// TIA Portal V15.1 export
// export: Created 2024-06-21T08:41:23.1994164Z, ExportSetting WithDefaults, DisplayName Totally Integrated Automation Portal, DisplayVersion V15.1 Update 5, DisplayName TIA Portal Openness, DisplayVersion V15.1 Update 5, DisplayName SINAMICS Startdrive Advanced, DisplayVersion V15.1, DisplayName G130, G150, S120, S150, SINAMICS MV, S210, DisplayVersion V15.1, DisplayName G110M, G120, G120C, G120D, G120P, DisplayVersion V15.1, DisplayName STEP 7 Professional, DisplayVersion V15.1 Update 5, DisplayName STEP 7 Safety, DisplayVersion V15.1, DisplayName WinCC Professional, DisplayVersion V15.1 Update 5, DisplayName SIMATIC Visualization Architect, DisplayVersion V15.1
FUNCTION "209210ZS01" : Void   // FC320, FBD
TITLE = 209210ZS01 Safety zone
{ S7_Optimized_Access := 'FALSE' }
AUTHOR : VCC
VERSION : 0.1
// stored: AutoNumber false, IsIECCheckEnabled false, SetENOAutomatically False, UDAEnableTagReadback false
   VAR_OUTPUT
      O_AlarmA : Bool;   // Alarm A
      O_AlarmB : Bool;   // Alarm B
      O_AlarmC : Bool;   // Alarm C
      O_AlarmD : Bool;   // Alarm D
      O_AlarmABCondition : Bool;   // Alarm AB Condition
      H_IAnim : Word;   // HMI Icon Animation
   END_VAR
BEGIN

REGION Network 1: **** 1 - Inputs **** HMI Reset / Start
   // Alarm Reset and Start from HMI
   // Note: connect signal "Safety not ok" from the FailSafe program
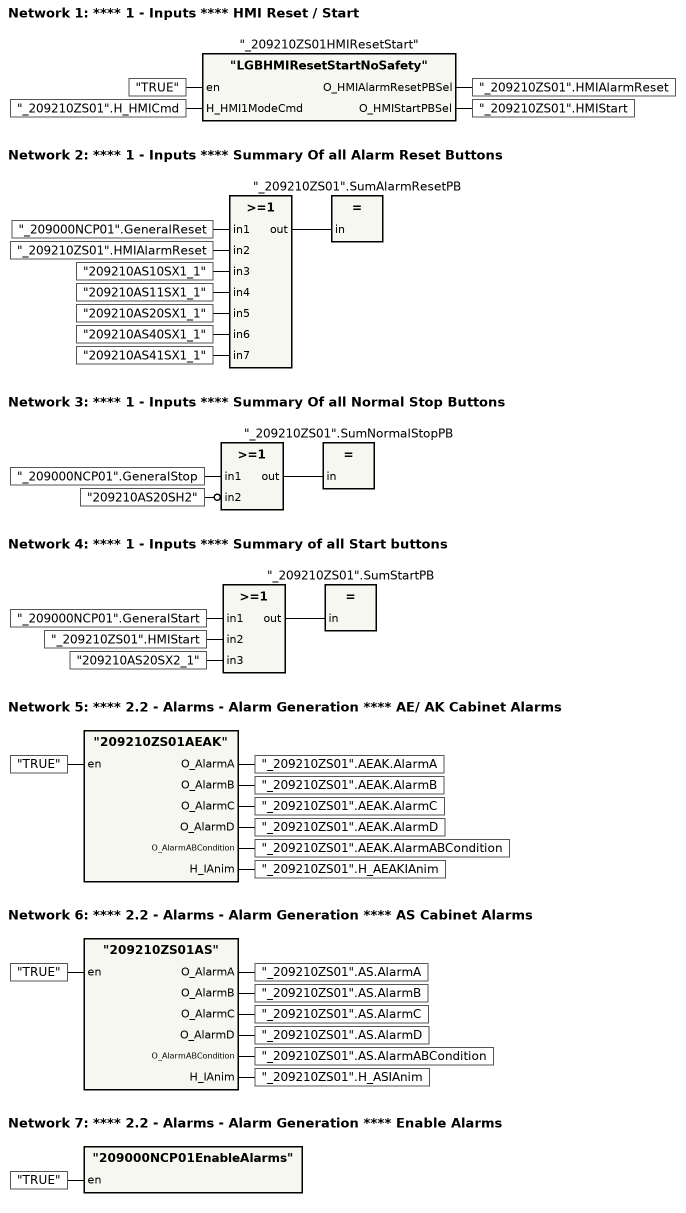
   IF "TRUE" THEN
       "_209210ZS01HMIResetStart"(H_HMI1ModeCmd := "_209210ZS01".H_HMICmd,   // "LGBHMIResetStartNoSafety"
                               O_HMIAlarmResetPBSel => "_209210ZS01".HMIAlarmReset,
                               O_HMIStartPBSel => "_209210ZS01".HMIStart);
   END_IF;
END_REGION

REGION Network 2: **** 1 - Inputs **** Summary Of all Alarm Reset Buttons
   // Summary Of all Alarm Reset Buttons accept the HMI's & Hardware panels Panels (Via LModeSelector)
   "_209210ZS01".SumAlarmResetPB := "_209000NCP01".GeneralReset OR "_209210ZS01".HMIAlarmReset OR "209210AS10SX1_1" OR "209210AS11SX1_1" OR "209210AS20SX1_1" OR "209210AS40SX1_1" OR "209210AS41SX1_1";
END_REGION

REGION Network 3: **** 1 - Inputs **** Summary Of all Normal Stop Buttons
   // Summary Of all Normal Stop Buttons accept the HMI's & Hardware panels Panels (Via LModeSelector)
   "_209210ZS01".SumNormalStopPB := "_209000NCP01".GeneralStop OR NOT "209210AS20SH2";
END_REGION

REGION Network 4: **** 1 - Inputs **** Summary of all Start buttons
   // Summary Of all Start Buttons accept the HMI's & Hardware panels Panels (Via LModeSelector)
   "_209210ZS01".SumStartPB := "_209000NCP01".GeneralStart OR "_209210ZS01".HMIStart OR "209210AS20SX2_1";
END_REGION

REGION Network 5: **** 2.2 - Alarms - Alarm Generation **** AE/ AK Cabinet Alarms
   // Cabinet Alarms
   IF "TRUE" THEN
       "209210ZS01AEAK"(O_AlarmA => "_209210ZS01".AEAK.AlarmA,
                        O_AlarmB => "_209210ZS01".AEAK.AlarmB,
                        O_AlarmC => "_209210ZS01".AEAK.AlarmC,
                        O_AlarmD => "_209210ZS01".AEAK.AlarmD,
                        O_AlarmABCondition => "_209210ZS01".AEAK.AlarmABCondition,
                        H_IAnim => "_209210ZS01".H_AEAKIAnim);
   END_IF;
END_REGION

REGION Network 6: **** 2.2 - Alarms - Alarm Generation **** AS Cabinet Alarms
   // AS Cabinet Alarms
   IF "TRUE" THEN
       "209210ZS01AS"(O_AlarmA => "_209210ZS01".AS.AlarmA,
                      O_AlarmB => "_209210ZS01".AS.AlarmB,
                      O_AlarmC => "_209210ZS01".AS.AlarmC,
                      O_AlarmD => "_209210ZS01".AS.AlarmD,
                      O_AlarmABCondition => "_209210ZS01".AS.AlarmABCondition,
                      H_IAnim => "_209210ZS01".H_ASIAnim);
   END_IF;
END_REGION

REGION Network 7: **** 2.2 - Alarms - Alarm Generation **** Enable Alarms
   IF "TRUE" THEN "209000NCP01EnableAlarms"(); END_IF;
END_REGION

REGION Network 8: **** 2.2 - Alarms - Alarm Generation **** Safety Alarms
   // Safety Alarms
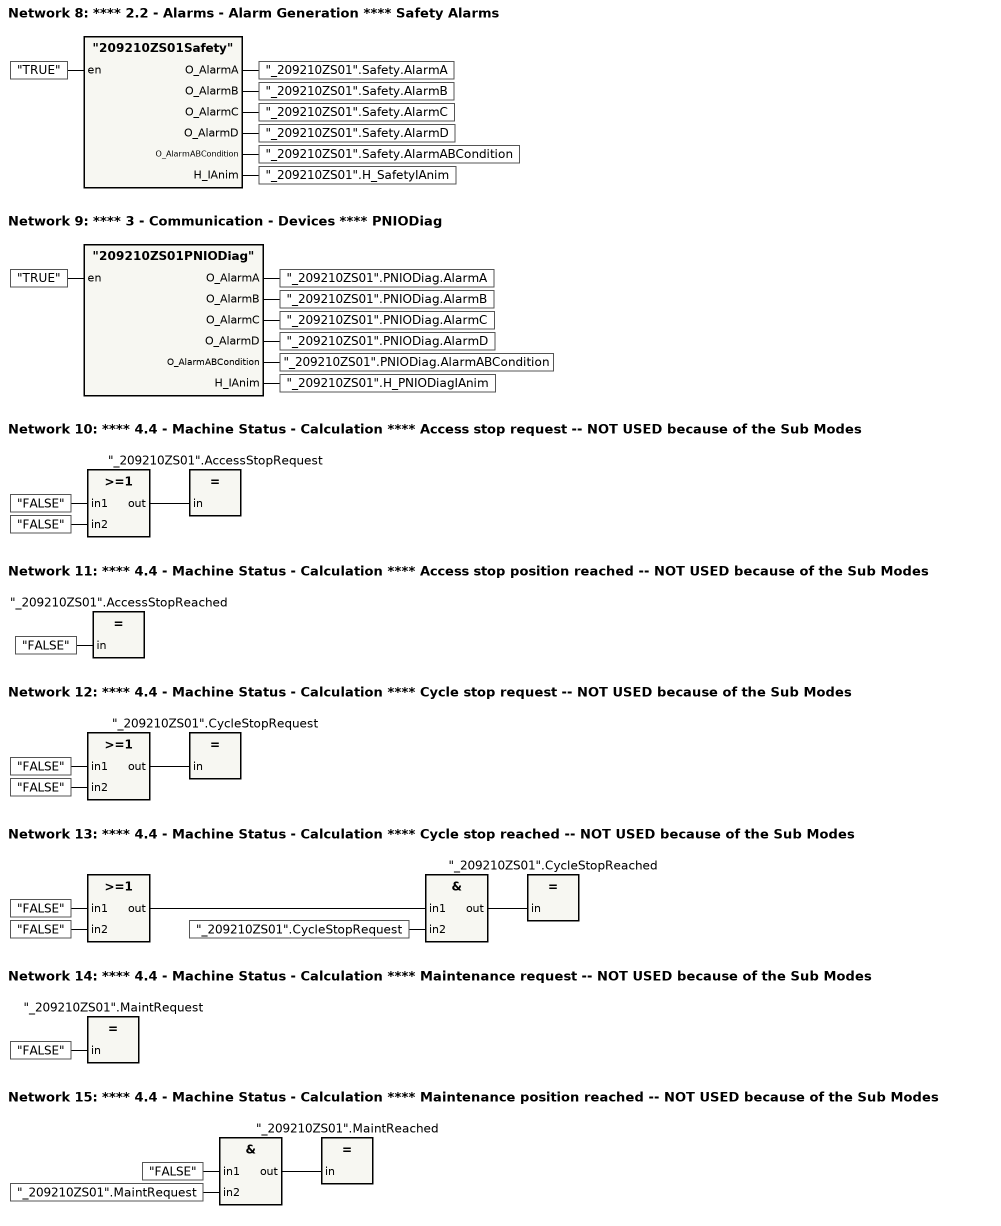
   IF "TRUE" THEN
       "209210ZS01Safety"(O_AlarmA => "_209210ZS01".Safety.AlarmA,
                          O_AlarmB => "_209210ZS01".Safety.AlarmB,
                          O_AlarmC => "_209210ZS01".Safety.AlarmC,
                          O_AlarmD => "_209210ZS01".Safety.AlarmD,
                          O_AlarmABCondition => "_209210ZS01".Safety.AlarmABCondition,
                          H_IAnim => "_209210ZS01".H_SafetyIAnim);
   END_IF;
END_REGION

REGION Network 9: **** 3 - Communication - Devices **** PNIODiag
   IF "TRUE" THEN
       "209210ZS01PNIODiag"(O_AlarmA => "_209210ZS01".PNIODiag.AlarmA,
                            O_AlarmB => "_209210ZS01".PNIODiag.AlarmB,
                            O_AlarmC => "_209210ZS01".PNIODiag.AlarmC,
                            O_AlarmD => "_209210ZS01".PNIODiag.AlarmD,
                            O_AlarmABCondition => "_209210ZS01".PNIODiag.AlarmABCondition,
                            H_IAnim => "_209210ZS01".H_PNIODiagIAnim);
   END_IF;
END_REGION

REGION Network 10: **** 4.4 - Machine Status - Calculation **** Access stop request -- NOT USED because of the Sub Modes
   // Access stop request
   "_209210ZS01".AccessStopRequest := "FALSE" OR "FALSE";
END_REGION

REGION Network 11: **** 4.4 - Machine Status - Calculation **** Access stop position reached -- NOT USED because of the Sub Modes
   // Access stop position reached
   "_209210ZS01".AccessStopReached := "FALSE";
END_REGION

REGION Network 12: **** 4.4 - Machine Status - Calculation **** Cycle stop request -- NOT USED because of the Sub Modes
   // Cycle stop request
   "_209210ZS01".CycleStopRequest := "FALSE" OR "FALSE";
END_REGION

REGION Network 13: **** 4.4 - Machine Status - Calculation **** Cycle stop reached -- NOT USED because of the Sub Modes
   // Cycle stop reached
   "_209210ZS01".CycleStopReached := ("FALSE" OR "FALSE") AND "_209210ZS01".CycleStopRequest;
END_REGION

REGION Network 14: **** 4.4 - Machine Status - Calculation **** Maintenance request -- NOT USED because of the Sub Modes
   // Maintenance request
   "_209210ZS01".MaintRequest := "FALSE";
END_REGION

REGION Network 15: **** 4.4 - Machine Status - Calculation **** Maintenance position reached -- NOT USED because of the Sub Modes
   // Maintenance position reached
   "_209210ZS01".MaintReached := "FALSE" AND "_209210ZS01".MaintRequest;
END_REGION

REGION Network 16: **** 4.5 - Machine status - Modes **** Modes Summary
   // Summary of all the modes in safety zone
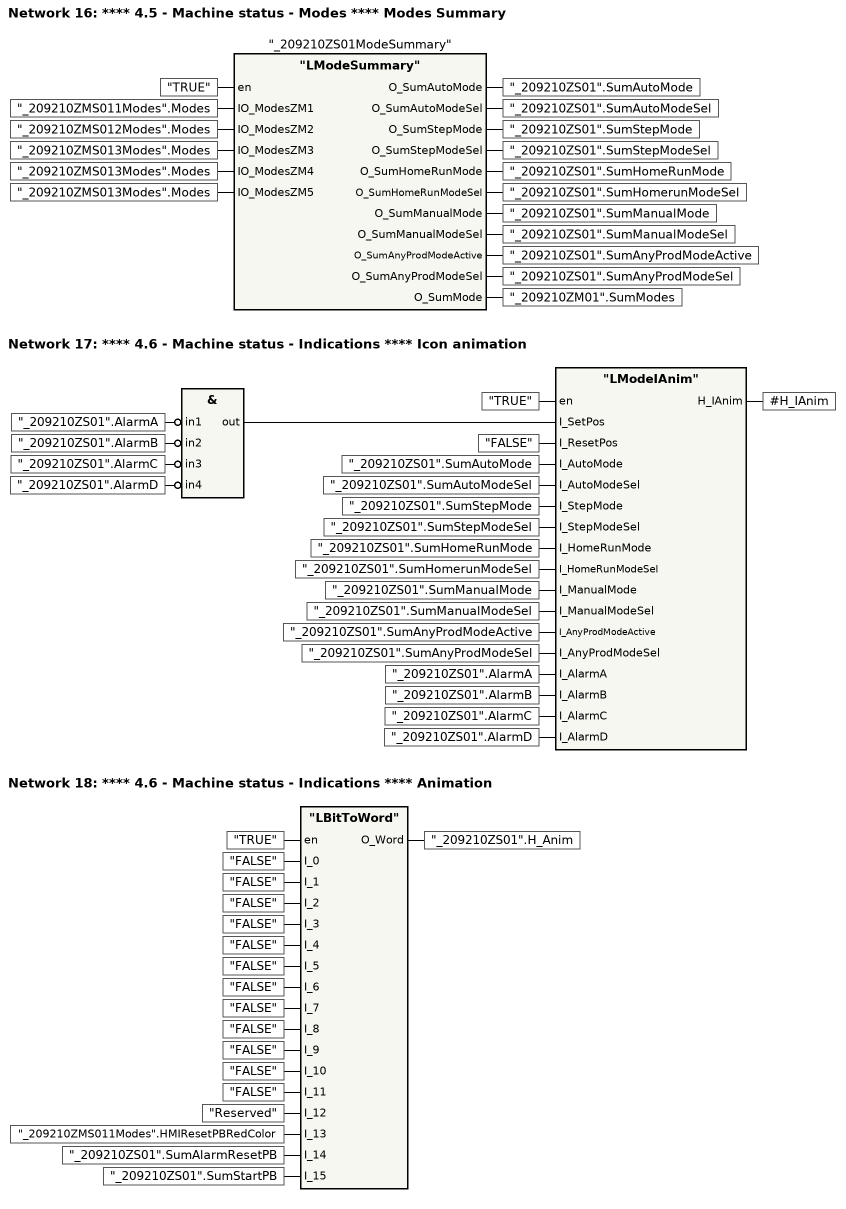
   IF "TRUE" THEN
       "_209210ZS01ModeSummary"(IO_ModesZM1 := "_209210ZMS011Modes".Modes,   // "LModeSummary"
                               IO_ModesZM2 := "_209210ZMS012Modes".Modes,
                               IO_ModesZM3 := "_209210ZMS013Modes".Modes,
                               IO_ModesZM4 := "_209210ZMS013Modes".Modes,
                               IO_ModesZM5 := "_209210ZMS013Modes".Modes,
                               O_SumAutoMode => "_209210ZS01".SumAutoMode,
                               O_SumAutoModeSel => "_209210ZS01".SumAutoModeSel,
                               O_SumStepMode => "_209210ZS01".SumStepMode,
                               O_SumStepModeSel => "_209210ZS01".SumStepModeSel,
                               O_SumHomeRunMode => "_209210ZS01".SumHomeRunMode,
                               O_SumHomeRunModeSel => "_209210ZS01".SumHomerunModeSel,
                               O_SumManualMode => "_209210ZS01".SumManualMode,
                               O_SumManualModeSel => "_209210ZS01".SumManualModeSel,
                               O_SumAnyProdModeActive => "_209210ZS01".SumAnyProdModeActive,
                               O_SumAnyProdModeSel => "_209210ZS01".SumAnyProdModeSel,
                               O_SumMode => "_209210ZM01".SumModes);
   END_IF;
END_REGION

REGION Network 17: **** 4.6 - Machine status - Indications **** Icon animation
   // Icon animation to WinCC
   IF "TRUE" THEN
       "LModeIAnim"(I_SetPos := NOT "_209210ZS01".AlarmA AND NOT "_209210ZS01".AlarmB AND NOT "_209210ZS01".AlarmC AND NOT "_209210ZS01".AlarmD,
                    I_ResetPos := "FALSE",
                    I_AutoMode := "_209210ZS01".SumAutoMode,
                    I_AutoModeSel := "_209210ZS01".SumAutoModeSel,
                    I_StepMode := "_209210ZS01".SumStepMode,
                    I_StepModeSel := "_209210ZS01".SumStepModeSel,
                    I_HomeRunMode := "_209210ZS01".SumHomeRunMode,
                    I_HomeRunModeSel := "_209210ZS01".SumHomerunModeSel,
                    I_ManualMode := "_209210ZS01".SumManualMode,
                    I_ManualModeSel := "_209210ZS01".SumManualModeSel,
                    I_AnyProdModeActive := "_209210ZS01".SumAnyProdModeActive,
                    I_AnyProdModeSel := "_209210ZS01".SumAnyProdModeSel,
                    I_AlarmA := "_209210ZS01".AlarmA,
                    I_AlarmB := "_209210ZS01".AlarmB,
                    I_AlarmC := "_209210ZS01".AlarmC,
                    I_AlarmD := "_209210ZS01".AlarmD,
                    H_IAnim => #H_IAnim);
   END_IF;
END_REGION

REGION Network 18: **** 4.6 - Machine status - Indications **** Animation
   // Animation
   IF "TRUE" THEN
       "LBitToWord"(I_0 := "FALSE",
                    I_1 := "FALSE",
                    I_2 := "FALSE",
                    I_3 := "FALSE",
                    I_4 := "FALSE",
                    I_5 := "FALSE",
                    I_6 := "FALSE",
                    I_7 := "FALSE",
                    I_8 := "FALSE",
                    I_9 := "FALSE",
                    I_10 := "FALSE",
                    I_11 := "FALSE",
                    I_12 := "Reserved",
                    I_13 := "_209210ZMS011Modes".HMIResetPBRedColor,
                    I_14 := "_209210ZS01".SumAlarmResetPB,
                    I_15 := "_209210ZS01".SumStartPB,
                    O_Word => "_209210ZS01".H_Anim);
   END_IF;
END_REGION

NETWORK
TITLE = **** 4.6 - Machine Status - Indications **** Animation DB number
// DB number
      OPN   "_209210ZS01";
      L     DBNO;
      T     "_209210ZS01".H_DBnr;

REGION Network 20: **** 7.3 - Submodule - Machine **** Zone Mode Conveyor
   // Zone Mode Conveyor
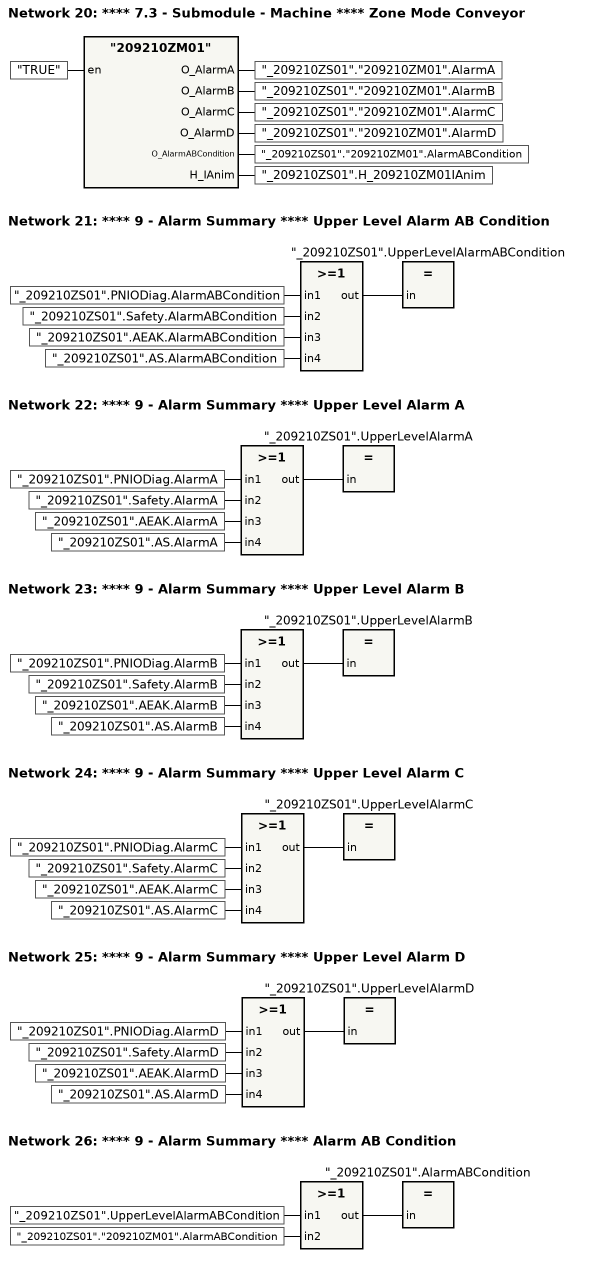
   IF "TRUE" THEN
       "209210ZM01"(O_AlarmA => "_209210ZS01"."209210ZM01".AlarmA,
                    O_AlarmB => "_209210ZS01"."209210ZM01".AlarmB,
                    O_AlarmC => "_209210ZS01"."209210ZM01".AlarmC,
                    O_AlarmD => "_209210ZS01"."209210ZM01".AlarmD,
                    O_AlarmABCondition => "_209210ZS01"."209210ZM01".AlarmABCondition,
                    H_IAnim => "_209210ZS01".H_209210ZM01IAnim);
   END_IF;
END_REGION

REGION Network 21: **** 9 - Alarm Summary **** Upper Level Alarm AB Condition
   // Upper Level Alarm AB condition
   "_209210ZS01".UpperLevelAlarmABCondition := "_209210ZS01".PNIODiag.AlarmABCondition OR "_209210ZS01".Safety.AlarmABCondition OR "_209210ZS01".AEAK.AlarmABCondition OR "_209210ZS01".AS.AlarmABCondition;
END_REGION

REGION Network 22: **** 9 - Alarm Summary **** Upper Level Alarm A
   // Upper Level Alarm A condition
   "_209210ZS01".UpperLevelAlarmA := "_209210ZS01".PNIODiag.AlarmA OR "_209210ZS01".Safety.AlarmA OR "_209210ZS01".AEAK.AlarmA OR "_209210ZS01".AS.AlarmA;
END_REGION

REGION Network 23: **** 9 - Alarm Summary **** Upper Level Alarm B
   // Upper Level Alarm B condition
   "_209210ZS01".UpperLevelAlarmB := "_209210ZS01".PNIODiag.AlarmB OR "_209210ZS01".Safety.AlarmB OR "_209210ZS01".AEAK.AlarmB OR "_209210ZS01".AS.AlarmB;
END_REGION

REGION Network 24: **** 9 - Alarm Summary **** Upper Level Alarm C
   // Upper Level Alarm C condition
   "_209210ZS01".UpperLevelAlarmC := "_209210ZS01".PNIODiag.AlarmC OR "_209210ZS01".Safety.AlarmC OR "_209210ZS01".AEAK.AlarmC OR "_209210ZS01".AS.AlarmC;
END_REGION

REGION Network 25: **** 9 - Alarm Summary **** Upper Level Alarm D
   // Upper Level Alarm D condition
   "_209210ZS01".UpperLevelAlarmD := "_209210ZS01".PNIODiag.AlarmD OR "_209210ZS01".Safety.AlarmD OR "_209210ZS01".AEAK.AlarmD OR "_209210ZS01".AS.AlarmD;
END_REGION

REGION Network 26: **** 9 - Alarm Summary **** Alarm AB Condition
   // Alarm AB condition
   "_209210ZS01".AlarmABCondition := "_209210ZS01".UpperLevelAlarmABCondition OR "_209210ZS01"."209210ZM01".AlarmABCondition;
END_REGION

REGION Network 27: **** 9 - Alarm Summary **** Alarm A
   // Summary of alarms A
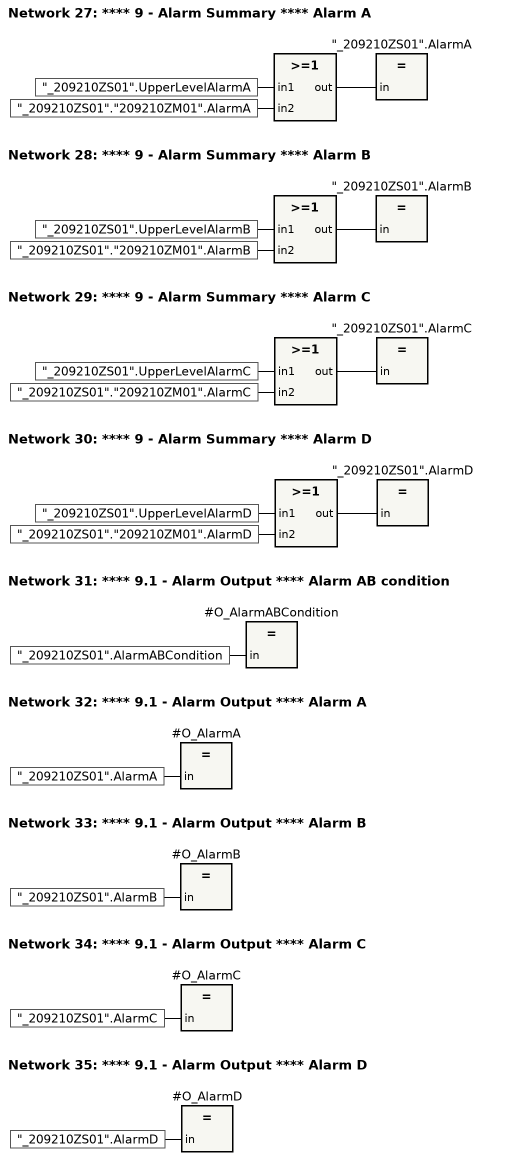
   "_209210ZS01".AlarmA := "_209210ZS01".UpperLevelAlarmA OR "_209210ZS01"."209210ZM01".AlarmA;
END_REGION

REGION Network 28: **** 9 - Alarm Summary **** Alarm B
   // Summary of alarms B
   "_209210ZS01".AlarmB := "_209210ZS01".UpperLevelAlarmB OR "_209210ZS01"."209210ZM01".AlarmB;
END_REGION

REGION Network 29: **** 9 - Alarm Summary **** Alarm C
   // Summary of alarms C
   "_209210ZS01".AlarmC := "_209210ZS01".UpperLevelAlarmC OR "_209210ZS01"."209210ZM01".AlarmC;
END_REGION

REGION Network 30: **** 9 - Alarm Summary **** Alarm D
   // Summary of alarms D
   "_209210ZS01".AlarmD := "_209210ZS01".UpperLevelAlarmD OR "_209210ZS01"."209210ZM01".AlarmD;
END_REGION

REGION Network 31: **** 9.1 - Alarm Output **** Alarm AB condition
   // Alarm AB condition
   #O_AlarmABCondition := "_209210ZS01".AlarmABCondition;
END_REGION

REGION Network 32: **** 9.1 - Alarm Output **** Alarm A
   // Output Alarm A
   #O_AlarmA := "_209210ZS01".AlarmA;
END_REGION

REGION Network 33: **** 9.1 - Alarm Output **** Alarm B
   // Output Alarm B
   #O_AlarmB := "_209210ZS01".AlarmB;
END_REGION

REGION Network 34: **** 9.1 - Alarm Output **** Alarm C
   // Output Alarm A
   #O_AlarmC := "_209210ZS01".AlarmC;
END_REGION

REGION Network 35: **** 9.1 - Alarm Output **** Alarm D
   // Output Alarm D
   #O_AlarmD := "_209210ZS01".AlarmD;
END_REGION

REGION Network 36: **** 9.2 - Alarm DWord**** Alarm To DWord
   // Alarm Word
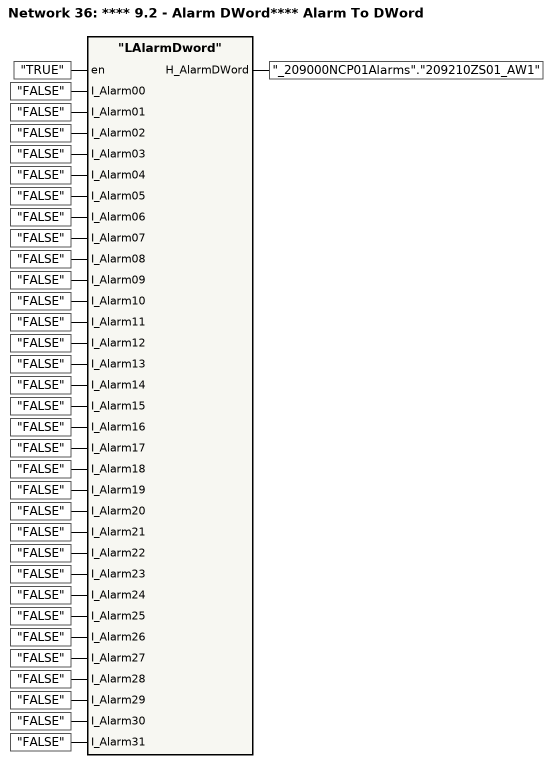
   IF "TRUE" THEN
       "LAlarmDword"(I_Alarm00 := "FALSE",
                     I_Alarm01 := "FALSE",
                     I_Alarm02 := "FALSE",
                     I_Alarm03 := "FALSE",
                     I_Alarm04 := "FALSE",
                     I_Alarm05 := "FALSE",
                     I_Alarm06 := "FALSE",
                     I_Alarm07 := "FALSE",
                     I_Alarm08 := "FALSE",
                     I_Alarm09 := "FALSE",
                     I_Alarm10 := "FALSE",
                     I_Alarm11 := "FALSE",
                     I_Alarm12 := "FALSE",
                     I_Alarm13 := "FALSE",
                     I_Alarm14 := "FALSE",
                     I_Alarm15 := "FALSE",
                     I_Alarm16 := "FALSE",
                     I_Alarm17 := "FALSE",
                     I_Alarm18 := "FALSE",
                     I_Alarm19 := "FALSE",
                     I_Alarm20 := "FALSE",
                     I_Alarm21 := "FALSE",
                     I_Alarm22 := "FALSE",
                     I_Alarm23 := "FALSE",
                     I_Alarm24 := "FALSE",
                     I_Alarm25 := "FALSE",
                     I_Alarm26 := "FALSE",
                     I_Alarm27 := "FALSE",
                     I_Alarm28 := "FALSE",
                     I_Alarm29 := "FALSE",
                     I_Alarm30 := "FALSE",
                     I_Alarm31 := "FALSE",
                     H_AlarmDWord => "_209000NCP01Alarms"."209210ZS01_AW1");
   END_IF;
END_REGION
END_FUNCTION
